INTERFACE ITF_InputDevice

METHOD ReadControlInputs : BOOL
VAR_INPUT
END_VAR
END_METHOD

END_INTERFACE

(* stored: Version 1.1.0.1, ProductVersion 3.1.4024.12
   Itf ITF_InputDevice: Id {d3365876-3dd2-4e76-8357-5b4cde50ea46}
   Method ReadControlInputs: Id {b75848ee-a316-47e6-9b12-5ccd6eb6d4b3} *)
